INTERFACE InterfaceSQLParameters

METHOD add_column : BOOL
VAR_INPUT
	sParaName : T_MaxString;
	eParaType : E_ExpParameterType;
	nParaSize : UDINT;
END_VAR
END_METHOD

PROPERTY cbParameters : UDINT
GET
END_GET
END_PROPERTY

PROPERTY column_num : UDINT
GET
END_GET
END_PROPERTY

PROPERTY insert_query_string : T_MaxString
GET
END_GET
END_PROPERTY

PROPERTY pParameters : PVOID
GET
END_GET
END_PROPERTY

PROPERTY table_name : T_MaxString
GET
END_GET
SET
END_SET
END_PROPERTY

END_INTERFACE

(* stored: Version 1.1.0.1, ProductVersion 3.1.4024.12
   Itf InterfaceSQLParameters: Id {9fc5e9e1-9a98-405b-a478-8d80d844167b}
   Method add_column: Id {5e59f425-57e0-4187-a42b-a5f60379a9e6}
   Property cbParameters: Id {ab51c17c-5edf-4b37-bc27-2f6b7e09c53a}
   Get Get: Id {0f52a21c-a803-4e13-b5fa-b7335458ea16}
   Property column_num: Id {a92aeef7-306b-4c0e-a6df-bae4fb57f6ea}
   Get Get: Id {e0008f07-4970-4d30-8aab-d3e5a1a92525}
   Property insert_query_string: Id {d9d90f1e-ac3a-4834-a8ad-26b226ba802e}
   Get Get: Id {e393c4b0-58cb-40d8-8644-3cf701f7ddda}
   Property pParameters: Id {aa8d4854-b052-47c7-856e-fb8c2666397b}
   Get Get: Id {911e03a4-b1e9-4b61-b9d3-7f26d4b3ddfd}
   Property table_name: Id {f3ae7ea5-76c1-443f-baaf-ef72a9115b5b}
   Get Get: Id {2fee4082-3d0e-4cd8-982a-23bcf1c98f91}
   Set Set: Id {c467b337-0daf-406c-8f65-7b8d8dccaec5} *)
